{attribute 'reflection'}
FUNCTION_BLOCK PUBLIC ABSTRACT FB_FunctionBase_WIthEvent EXTENDS FB_Base_WithEvent
VAR_INPUT
	bSafetyOk	: BOOL 		:= TRUE 				; // Module can operate safely [default true]
END_VAR
VAR_OUTPUT
	sActiveState	: STRING 		:= 'Idle'	; // active state of device 
	bManual			: BOOL 			:= FALSE 	; // device is in manual mode
	bIsSafe			: BOOL 			:= FALSE	; // Device is locked and safe
	bHeld			: BOOL 			:= FALSE 	; // Function is held
	bBlockedCommand	: BOOL 			:= FALSE 	; // a device command is blocked because of collision detect 
END_VAR
VAR
	bCmdManual 		: BOOL			:= FALSE	; // manual commands enabled control functions (thus disable automatic)
END_VAR

SUPER^();

// Communicate active state
IF NOT bSafetyOk THEN 
	sActiveState := 'Safety not ok';
ELSIF bErrorActive THEN 
	sActiveState := 'Error is active';
ELSIF NOT bInitOk THEN 
	sActiveState := 'Not initialized';
ELSIF bManual THEN 
	sActiveState := 'Operational';
END_IF 

// check for manual command mode
bManual := bCmdManual ;

// Execute device functions
IF bInitOk THEN  
	ExecMachineSafety();
	ExecDevFunctions();
END_IF

// Set fault if commands are blocked
IF bBlockedCommand THEN 
	fbEvent.CmdAddEvent( Event := TC_EVENTS.StateMessages.FunctionsIsBlocked);
END_IF

METHOD PUBLIC CmdHold : BOOL
VAR_INPUT
END_VAR
bHeld 	:= TRUE ;
CmdHold := bHeld ;
END_METHOD

METHOD PUBLIC CmdManual : BOOL
VAR_INPUT
END_VAR
bCmdManual := true ;
END_METHOD

METHOD PUBLIC CmdSafeStop : BOOL
VAR_INPUT
END_VAR
// check if device is safe
bIsSafe 	:= NOT bEnable ;
CmdSafeStop := bIsSafe ;
END_METHOD

METHOD PROTECTED ExecDevFunctions : BOOL
VAR_INPUT
END_VAR
END_METHOD

METHOD PROTECTED ExecMachineSafety : BOOL
VAR_INPUT
END_VAR
END_METHOD

END_FUNCTION_BLOCK

(* stored: Version 1.1.0.1, ProductVersion 3.1.4024.9
   POU FB_FunctionBase_WIthEvent: Id {0140c1b6-1d19-4ea0-a668-c0411892cb34}, SpecialFunc None
   Method CmdHold: Id {6f5da2de-a0c9-45a9-97e4-4c7c0bf3aed8}
   Method CmdManual: Id {db0662d6-d805-4046-ab9d-4a7e60512933}
   Method CmdSafeStop: Id {b6bb3a29-0ede-44ee-b37b-c4108cb4759e}
   Method ExecDevFunctions: Id {7fc95b8e-87fc-4948-aad6-2622ac8b1ac8}
   Method ExecMachineSafety: Id {b5f44ac6-135f-4436-8d72-9ac63890bc3c} *)
